INTERFACE I_RpcArguments

METHOD NoReturnValue : I_RpcInvoke
VAR_INPUT
END_VAR
END_METHOD

METHOD ReturnValue : I_RpcInvoke
VAR_INPUT
	anyRetVal	: ANY;
END_VAR
END_METHOD

METHOD VarInOut : I_RpcArguments
VAR_INPUT
	anyArg	: ANY;
END_VAR
END_METHOD

METHOD VarInput : I_RpcArguments
VAR_INPUT
	anyArg	: ANY;
END_VAR
END_METHOD

METHOD VarOutput : I_RpcArguments
VAR_INPUT
	anyArg	: ANY;
END_VAR
END_METHOD

END_INTERFACE

(* stored: Version 1.1.0.1, ProductVersion 3.1.4024.12
   Itf I_RpcArguments: Id {f01db549-96f9-4574-a861-747d1e7a3b06}
   Method NoReturnValue: Id {fe67e016-bc9b-4392-8c32-1218f7b4b53d}
   Method ReturnValue: Id {58afd851-a822-4452-8c2b-a0e87f1e7b8f}
   Method VarInOut: Id {aaeb6169-ca97-467d-b043-1dc6a7ed05a3}
   Method VarInput: Id {968e2530-cbac-40a7-82b0-950291c5a931}
   Method VarOutput: Id {b0441363-d524-4a34-8dcc-abd11b12ecea} *)
